Staubli VAL3: HerePoint.pgx

public program HerePoint(num x_nIndex)
  local tool l_tTool
  local point l_pHere
  local frame l_fFrame
  local num i
  local num l_nIndex
  local num l_nSize
begin
  //
  // take the point
  //
  // tool
  call tcp:getTool(l_tTool,pEditPoint.nIndexTool)
  // here
  l_pHere=here(l_tTool,pEditPoint.fFrame)
  resetMotion()
  // save the trsf
  pEditPoint.tData[x_nIndex].pPoint.trsf=l_pHere.trsf
  // check the moveType to save the config
  if pEditPoint.tData[x_nIndex].tSuper.moveType==0
    pEditPoint.tData[x_nIndex].pPoint.config=l_pHere.config
  endIf
end
